TYPE EL6021_Data :
STRUCT
	{attribute addProperty Name "COM TxPDO-Map Inputs"}
	COM_TxPDO_Map_Inputs : EL6021_COM_Inputs;
	{attribute addProperty Name "COM RxPDO-Map Outputs"}
	COM_RxPDO_Map_Outputs : EL6021_COM_Outputs;
END_STRUCT
END_TYPE

(* stored: Version 1.1.0.1, ProductVersion 3.1.4024.9
   DUT EL6021_Data: Id {6ae7d704-5ebe-0c11-070e-0c34e91d90a7} *)
